{attribute addProperty BoxType "EL6900-0000-0016"}
{attribute addProperty Id "DEVICE_InputsAT %I*DEVICE_Inputs_3148493E4860DEVICE_OutputsAT %Q*DEVICE_Outputs_734938A41620WcStateAT %I*WcState_98A4DF7520.250InfoDataAT %I*InfoData_BC63D37F80100"}
{attribute addProperty CRC "227112445"}
{attribute addProperty SizeInBites "146"}
{attribute addProperty SizeInBytes "18.25"}
TYPE EL6900_4A623936 :
STRUCT
	{attribute addProperty Name "DEVICE_Inputs"}
	DEVICE_Inputs : DEVICE_Inputs_3148493E;
	{attribute addProperty Name "DEVICE_Outputs"}
	DEVICE_Outputs : DEVICE_Outputs_734938A4;
	{attribute addProperty Name "WcState"}
	WcState : WcState_98A4DF75;
	{attribute addProperty Name "InfoData"}
	InfoData : InfoData_BC63D37F;
END_STRUCT
END_TYPE

(* stored: Version 1.2.0.0, ProductVersion 3.1.4024.9
   DUT EL6900_4A623936: Id {cc8eda20-0ba4-423d-b399-7de772fba984} *)
